LIN {X 0,Y 112.602,Z 689.131,A -85,B 0,C 180,E1 -30780.001,E2 -30780.001} C_VEL
LIN {X 0,Y 107.319,Z 691.975,A -85,B 0,C 180,E1 -30780.555,E2 -30780.555} C_VEL
LIN {X 0,Y 96.352,Z 697.207,A -85,B 0,C 180,E1 -30781.185,E2 -30781.185} C_VEL
LIN {X 0,Y 85.017,Z 701.685,A -85,B 0,C 180,E1 -30781.632,E2 -30781.632} C_VEL
LIN {X 0,Y 73.474,Z 705.296,A -85,B 0,C 180,E1 -30782.713,E2 -30782.713} C_VEL
LIN {X 0,Y 67.735,Z 706.633,A -85,B 0,C 180,E1 -30783.896,E2 -30783.896} C_VEL
LIN {X 0,Y 56.694,Z 708.733,A -85,B 0,C 180,E1 -30787.414,E2 -30787.414} C_VEL
LIN {X 0,Y 43.419,Z 710.237,A -85,B 0,C 180,E1 -30793.809,E2 -30793.809} C_VEL
LIN {X 0,Y 31.072,Z 710.589,A -85,B 0,C 180,E1 -30805.227,E2 -30805.227} C_VEL
LIN {X 0,Y 21.126,Z 709.778,A -85,B 0,C 180,E1 -30828.303,E2 -30828.303} C_VEL
LIN {X 0,Y 17.791,Z 707.877,A -85,B 0,C 180,E1 -30870.009,E2 -30870.009} C_VEL
LIN {X 0,Y 23.974,Z 704.844,A -85,B 0,C 180,E1 -30905.902,E2 -30905.902} C_VEL
LIN {X 0,Y 34.793,Z 700.645,A -85,B 0,C 180,E1 -30923.904,E2 -30923.904} C_VEL
LIN {X 0,Y 47.156,Z 695.178,A -85,B 0,C 180,E1 -30933.412,E2 -30933.412} C_VEL
LIN {X 0,Y 60.174,Z 688.261,A -85,B 0,C 180,E1 -30939.129,E2 -30939.129} C_VEL
LIN {X 0,Y 71.8,Z 680.893,A -85,B 0,C 180,E1 -30942.626,E2 -30942.626} C_VEL
LIN {X 0,Y 83.578,Z 672.021,A -85,B 0,C 180,E1 -30945.247,E2 -30945.247} C_VEL
LIN {X 0,Y 95.44,Z 661.343,A -85,B 0,C 180,E1 -30947.344,E2 -30947.344} C_VEL
LIN {X 0,Y 105.621,Z 650.419,A -85,B 0,C 180,E1 -30948.95,E2 -30948.95} C_VEL
LIN {X 0,Y 114.965,Z 638.478,A -85,B 0,C 180,E1 -30950.315,E2 -30950.315} C_VEL
LIN {X 0,Y 123.521,Z 625.292,A -85,B 0,C 180,E1 -30951.335,E2 -30951.335} C_VEL
LIN {X 0,Y 131.228,Z 610.533,A -85,B 0,C 180,E1 -30952.211,E2 -30952.211} C_VEL
LIN {X 0,Y 137.196,Z 595.922,A -85,B 0,C 180,E1 -30952.921,E2 -30952.921} C_VEL
LIN {X 0,Y 141.47,Z 582.197,A -85,B 0,C 180,E1 -30953.494,E2 -30953.494} C_VEL
LIN {X 0,Y 144.889,Z 566.394,A -85,B 0,C 180,E1 -30953.909,E2 -30953.909} C_VEL
LIN {X 0,Y 145.85,Z 559.827,A -85,B 0,C 180,E1 -30954.122,E2 -30954.122} C_VEL
LIN {X 0,Y 145.892,Z 559.552,A -85,B 0,C 180,E1 -30954.732,E2 -30954.732} C_VEL
LIN {X 0,Y 143.283,Z 574.841,A -85,B 0,C 180,E1 -30954.898,E2 -30954.898} C_VEL
LIN {X 0,Y 139.223,Z 590.241,A -85,B 0,C 180,E1 -30955.11,E2 -30955.11} C_VEL
LIN {X 0,Y 133.533,Z 605.838,A -85,B 0,C 180,E1 -30955.343,E2 -30955.343} C_VEL
LIN {X 0,Y 126.88,Z 619.972,A -85,B 0,C 180,E1 -30955.583,E2 -30955.583} C_VEL
LIN {X 0,Y 120.677,Z 630.75,A -85,B 0,C 180,E1 -30955.805,E2 -30955.805} C_VEL
LIN {X 0,Y 112.702,Z 642.546,A -85,B 0,C 180,E1 -30956.147,E2 -30956.147} C_VEL
LIN {X 0,Y 103.856,Z 653.624,A -85,B 0,C 180,E1 -30956.509,E2 -30956.509} C_VEL
LIN {X 0,Y 93.234,Z 664.888,A -85,B 0,C 180,E1 -30957.176,E2 -30957.176} C_VEL
LIN {X 0,Y 82.616,Z 674.506,A -85,B 0,C 180,E1 -30958.299,E2 -30958.299} C_VEL
LIN {X 0,Y 70.281,Z 683.93,A -85,B 0,C 180,E1 -30959.999,E2 -30959.999} C_VEL
LIN {X 0,Y 58.038,Z 691.788,A -85,B 0,C 180,E1 -30962.507,E2 -30962.507} C_VEL
LIN {X 0,Y 45.981,Z 698.331,A -85,B 0,C 180,E1 -30966.517,E2 -30966.517} C_VEL
LIN {X 0,Y 32.736,Z 704.404,A -85,B 0,C 180,E1 -30974.951,E2 -30974.951} C_VEL
LIN {X 0,Y 23.713,Z 708.066,A -85,B 0,C 180,E1 -30987.225,E2 -30987.225} C_VEL
LIN {X 0,Y 15.678,Z 711.759,A -85,B 0,C 180,E1 -31023.695,E2 -31023.695} C_VEL
LIN {X 0,Y 15.524,Z 713.092,A -85,B 0,C 180,E1 -31049.99,E2 -31049.99} C_VEL
LIN {X 0,Y 16.458,Z 713.85,A -85,B 0,C 180,E1 -31081.358,E2 -31081.358} C_VEL
LIN {X 0,Y 23.834,Z 714.074,A -85,B 0,C 180,E1 -31112.189,E2 -31112.189} C_VEL
LIN {X 0,Y 36.034,Z 713.349,A -85,B 0,C 180,E1 -31127.185,E2 -31127.185} C_VEL
LIN {X 0,Y 49.433,Z 711.494,A -85,B 0,C 180,E1 -31134.341,E2 -31134.341} C_VEL
LIN {X 0,Y 63.278,Z 708.531,A -85,B 0,C 180,E1 -31138.217,E2 -31138.217} C_VEL
LIN {X 0,Y 77.306,Z 704.444,A -85,B 0,C 180,E1 -31140.512,E2 -31140.512} C_VEL
LIN {X 0,Y 77.334,Z 704.261,A -85,B 0,C 180,E1 -31141.627,E2 -31141.627} C_VEL
LIN {X 0,Y 67.735,Z 706.633,A -85,B 0,C 180,E1 -31143.896,E2 -31143.896} C_VEL
LIN {X 0,Y 62.062,Z 707.917,A -85,B 0,C 180,E1 -31144.892,E2 -31144.892} C_VEL
LIN {X 0,Y 52.319,Z 709.794,A -85,B 0,C 180,E1 -31145.043,E2 -31145.043} C_VEL
LIN {X 0,Y 42.492,Z 711.133,A -85,B 0,C 180,E1 -31145.175,E2 -31145.175} C_VEL
LIN {X 0,Y 36.72,Z 711.51,A -85,B 0,C 180,E1 -31146.891,E2 -31146.891} C_VEL
LIN {X 0,Y 22.357,Z 711.362,A -85,B 0,C 180,E1 -31159.453,E2 -31159.453} C_VEL
LIN {X 0,Y 11.973,Z 710.059,A -85,B 0,C 180,E1 -31194.074,E2 -31194.074} C_VEL
LIN {X 0,Y 13.546,Z 707.641,A -85,B 0,C 180,E1 -31261.265,E2 -31261.265} C_VEL
LIN {X 0,Y 24.797,Z 704.067,A -85,B 0,C 180,E1 -31288.249,E2 -31288.249} C_VEL
LIN {X 0,Y 37.753,Z 699.321,A -85,B 0,C 180,E1 -31298.564,E2 -31298.564} C_VEL
LIN {X 0,Y 51.238,Z 693.204,A -85,B 0,C 180,E1 -31303.777,E2 -31303.777} C_VEL
LIN {X 0,Y 64.896,Z 685.549,A -85,B 0,C 180,E1 -31307.079,E2 -31307.079} C_VEL
LIN {X 0,Y 76.755,Z 677.551,A -85,B 0,C 180,E1 -31309.23,E2 -31309.23} C_VEL
LIN {X 0,Y 88.972,Z 667.664,A -85,B 0,C 180,E1 -31310.88,E2 -31310.88} C_VEL
LIN {X 0,Y 99.338,Z 657.677,A -85,B 0,C 180,E1 -31312.086,E2 -31312.086} C_VEL
LIN {X 0,Y 99.207,Z 657.896,A -85,B 0,C 180,E1 -31312.651,E2 -31312.651} C_VEL
LIN {X 0,Y 88.506,Z 668.375,A -85,B 0,C 180,E1 -31313.022,E2 -31313.022} C_VEL
LIN {X 0,Y 75.851,Z 678.774,A -85,B 0,C 180,E1 -31313.77,E2 -31313.77} C_VEL
LIN {X 0,Y 63.519,Z 687.224,A -85,B 0,C 180,E1 -31314.752,E2 -31314.752} C_VEL
LIN {X 0,Y 49.278,Z 695.31,A -85,B 0,C 180,E1 -31316.729,E2 -31316.729} C_VEL
LIN {X 0,Y 35.144,Z 701.798,A -85,B 0,C 180,E1 -31320.584,E2 -31320.584} C_VEL
LIN {X 0,Y 21.393,Z 706.855,A -85,B 0,C 180,E1 -31329.714,E2 -31329.714} C_VEL
LIN {X 0,Y 9.343,Z 710.788,A -85,B 0,C 180,E1 -31368.768,E2 -31368.768} C_VEL
LIN {X 0,Y 8.336,Z 711.968,A -85,B 0,C 180,E1 -31409.981,E2 -31409.981} C_VEL
LIN {X 0,Y 10.569,Z 712.706,A -85,B 0,C 180,E1 -31458.334,E2 -31458.334} C_VEL
LIN {X 0,Y 21.445,Z 713.025,A -85,B 0,C 180,E1 -31489.427,E2 -31489.427} C_VEL
LIN {X 0,Y 35.145,Z 712.342,A -85,B 0,C 180,E1 -31498.742,E2 -31498.742} C_VEL
LIN {X 0,Y 47.731,Z 710.749,A -85,B 0,C 180,E1 -31502.397,E2 -31502.397} C_VEL
LIN {X 0,Y 36.72,Z 711.51,A -85,B 0,C 180,E1 -31506.891,E2 -31506.891} C_VEL
LIN {X 0,Y 30.501,Z 711.76,A -85,B 0,C 180,E1 -31509.488,E2 -31509.488} C_VEL
LIN {X 0,Y 19.809,Z 711.819,A -85,B 0,C 180,E1 -31511.988,E2 -31511.988} C_VEL
LIN {X 0,Y 11.242,Z 711.454,A -85,B 0,C 180,E1 -31516.022,E2 -31516.022} C_VEL
LIN {X 0,Y 4.581,Z 710.667,A -85,B 0,C 180,E1 -31543.217,E2 -31543.217} C_VEL
LIN {X 0,Y 3.987,Z 710.441,A -85,B 0,C 180,E1 -31555.067,E2 -31555.067} C_VEL
LIN {X 0,Y 8.35,Z 708.773,A -85,B 0,C 180,E1 -31647.347,E2 -31647.347} C_VEL
LIN {X 0,Y 21.919,Z 705.25,A -85,B 0,C 180,E1 -31664.153,E2 -31664.153} C_VEL
LIN {X 0,Y 28.843,Z 703.056,A -85,B 0,C 180,E1 -31667.089,E2 -31667.089} C_VEL
LIN {X 0,Y 28.598,Z 703.263,A -85,B 0,C 180,E1 -31669.448,E2 -31669.448} C_VEL
LIN {X 0,Y 14.202,Z 707.697,A -85,B 0,C 180,E1 -31671.848,E2 -31671.848} C_VEL
LIN {X 0,Y 1.155,Z 710.844,A -85,B 0,C 180,E1 -31769.866,E2 -31769.866} C_VEL
LIN {X 0,Y 7.202,Z 711.56,A -85,B 0,C 180,E1 -31860.014,E2 -31860.014} C_VEL
LIN {X 0,Y 12.708,Z 711.863,A -85,B 0,C 180,E1 -31865.849,E2 -31865.849} C_VEL
LIN {X 0,Y 7.487,Z 711.146,A -85,B 0,C 180,E1 -31880.225,E2 -31880.225} C_VEL
LIN {X 0,Y 3.987,Z 710.441,A -85,B 0,C 180,E1 -31915.067,E2 -31915.067} C_VEL
LIN {X 0,Y 3.987,Z 710.441,A -85,B 0,C 180,E1 -31915.067,E2 -31915.067}

QRS_NEXT_CUT()

QRS_NEXT()
QRS_HOME()

END
